ABB RobotStudio station: Apartado4.rspag

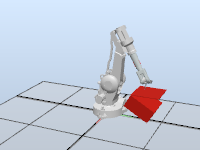
--- station ---
Station Práctica_1_casa (saved by RobotStudio 7.0.8746.631)
Controller IRB_2400_12kg_1.55m
  mechanical unit ROB_1: IRB2400_10_150__02, 6 joints, base frame (0, 0, 0) mm
Layout (positions relative to the parent item):
  - IRB2400_10_150__02 [mechanism, from Robots\IRB2400_10_150_G_02.rslib] at (0, 0, 0) mm; joint values [1.6074, 0.1285, 1.0857, 1.3381, 1.0961, 3.693] (rad or m)
  - Inclinado [part] at (-150, 550, 100) mm, rotated rx 0 ry 30 rz 90 deg
  - Garra_puntero_simple [smart component, from Libraries\Garra_puntero_simple.rslib] at (-97.85, 661.37, 666.74) mm, rotated rx -180 ry 60 rz 0 deg
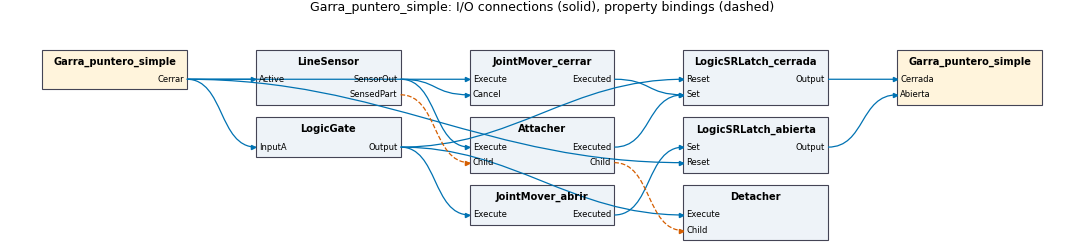
      connections:
        Garra_puntero_simple.Cerrar -> LineSensor.Active
        LineSensor.SensorOut -> Attacher.Execute
        Garra_puntero_simple.Cerrar -> JointMover_cerrar.Execute
        LineSensor.SensorOut -> JointMover_cerrar.Cancel
        Garra_puntero_simple.Cerrar -> LogicGate.InputA
        LogicGate.Output -> Detacher.Execute
        LogicGate.Output -> JointMover_abrir.Execute
        LogicGate.Output -> LogicSRLatch_cerrada.Reset
        LogicSRLatch_cerrada.Output -> Garra_puntero_simple.Cerrada
        JointMover_abrir.Executed -> LogicSRLatch_abierta.Set
        Garra_puntero_simple.Cerrar -> LogicSRLatch_abierta.Reset
        LogicSRLatch_abierta.Output -> Garra_puntero_simple.Abierta
        Attacher.Executed -> LogicSRLatch_cerrada.Set
        JointMover_cerrar.Executed -> LogicSRLatch_cerrada.Set
        LineSensor.SensedPart => Attacher.Child
        Attacher.Child => Detacher.Child
    - LineSensor [smart component, from Components\LineSensor.rslib] at (0, 60, 0) mm
        properties: Start=[0 -0.0595 0.149]; End=[3.45126646034193E-31 -0.0595 0.045]; Radius=0.0001; SensedPart=(none); SensedPoint=[0 0 0]
      - _sensorPart_ [part]
    - Attacher [smart component, from Components\Attacher.rslib]
        properties: Parent=Mecanismo_garra_puntero_simple; Flange=0; Child=(none); Mount=false; Offset=[0 0 0]; Orientation=[0 0 0]
    - Detacher [smart component, from Components\Detacher.rslib]
        properties: Child=Mecanismo_garra_puntero_simple; KeepPosition=true
    - JointMover_cerrar [smart component, from Components\JointMover.rslib]
        properties: Mechanism=Mecanismo_garra_puntero_simple; Relative=false; Duration=0.5; J1=0
    - LogicGate [smart component, from Components\LogicGate.rslib]
        properties: Operator=NOT; Delay=0
    - JointMover_abrir [smart component, from Components\JointMover.rslib]
        properties: Mechanism=Mecanismo_garra_puntero_simple; Relative=false; Duration=0.5; J1=0.06
    - LogicSRLatch_cerrada [smart component, from Components\LogicSRLatch.rslib]
    - LogicSRLatch_abierta [smart component, from Components\LogicSRLatch.rslib]
    - Mecanismo_garra_puntero_simple [mechanism, from Libraries\Garra_puntero_simple.rslib] at (0, 0, 0) mm; joint values [0.06] (rad or m)
Attachment: LineSensor is attached to Mecanismo_garra_puntero_simple / Dedp_1
Attachment: Garra_puntero_simple is attached to IRB2400_10_150__02 / Link6
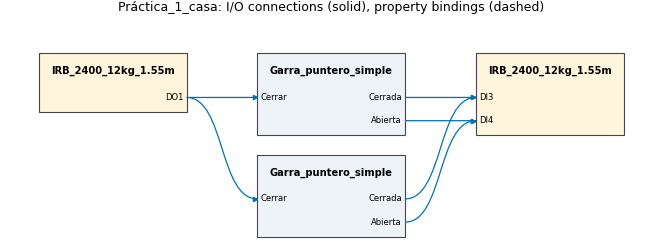
Station logic (signal -> signal, property => property):
  Garra_puntero_simple.Cerrada -> IRB_2400_12kg_1.55m.DI3
  Garra_puntero_simple.Abierta -> IRB_2400_12kg_1.55m.DI4
  IRB_2400_12kg_1.55m.DO1 -> Garra_puntero_simple.Cerrar
  Garra_puntero_simple.Cerrada -> IRB_2400_12kg_1.55m.DI3
  Garra_puntero_simple.Abierta -> IRB_2400_12kg_1.55m.DI4
  IRB_2400_12kg_1.55m.DO1 -> Garra_puntero_simple.Cerrar

--- Backups/IRB_2400_12kg_1.55m/RAPID/TASK1/PROGMOD/Module1.mod ---
MODULE Module1
    PERS tooldata Garra_TCP:=[TRUE,[[0,0,150],[0,1,0,0]],[1,[0,0,10],[1,0,0,0],0,0,0]];
    PERS tooldata Puntero_TCP:=[TRUE,[[150,0,30],[0.707106781,0,-0.707106781,0]],[1,[0,0,10],[1,0,0,0],0,0,0]];
    CONST confdata config_fun:=[0,0,0,0];
    CONST confdata config_fuf:=[0,0,0,1];
    CONST extjoint ejes_externos:=[9E+09,9E+09,9E+09,9E+09,9E+09,9E+09];
    CONST jointtarget casa:=[[0,0,0,0,0,0],ejes_externos];
    CONST num distancia:=150;
    TASK PERS wobjdata plano_trazado:=[FALSE,TRUE,"",[[101.172,952.795,450.836],[2.49104E-07,0,0,1]],[[0,0,0],[1,0,0,0]]];

    VAR intnum emergencia;

    PROC Pinta_cuadrado(robtarget centro, PERS wobjdata objeto_trabajo, PERS tooldata tool)
        VAR robtarget Paprox;
        VAR robtarget P1;
        VAR robtarget P2;
        VAR robtarget P3;
        VAR robtarget P4;

        Paprox:= RelTool (centro, 0, 0, 50);
        MoveJ Paprox, v500, fine, tool\WObj:=objeto_trabajo;

        P1:= RelTool (centro, 50, 50, 0);
        MoveL P1, v500, fine, tool\WObj:=objeto_trabajo;

        P2:= RelTool (centro, 50, -50, 0);
        MoveL P2, v500, fine, tool\WObj:=objeto_trabajo;

        P3:= RelTool (centro, -50, -50, 0);
        MoveL P3, v500, fine, tool\WObj:=objeto_trabajo;

        P4:= RelTool (centro, -50, 50, 0);
        MoveL P4, v500, fine, tool\WObj:=objeto_trabajo;

        !Move to complete square
        MoveL P1, v500, fine, tool\WObj:=objeto_trabajo;

        !Move to approximation position
        MoveL Paprox, v500, fine, tool\WObj:=objeto_trabajo;
    ENDPROC

    PROC Pinta_circunferencia(robtarget centro, PERS wobjdata objeto_trabajo, PERS tooldata tool)
        VAR robtarget Paprox;
        VAR robtarget P1;
        VAR robtarget P2;
        VAR robtarget P3;
        VAR robtarget P4;

        Paprox:= RelTool (centro, 0, 0, 50);
        MoveJ Paprox, v500, fine, tool\WObj:=objeto_trabajo;

        P1:= RelTool (centro, 0, 100*Sqrt(2), 0);
        P2:= RelTool (centro, 100*Sqrt(2), 0, 0);
        P3:= RelTool (centro, 0, -100*Sqrt(2), 0);
        P4:= RelTool (centro, -100*Sqrt(2), 0, 0);

        MoveL P1, v500, fine, tool\WObj:=objeto_trabajo;
        MoveC P2, P3, v500, fine, tool\WObj:=objeto_trabajo;
        MoveC P4, P1, v500, fine, tool\WObj:=objeto_trabajo;

        MoveJ Paprox, v500, fine, tool\WObj:=objeto_trabajo;

	ENDPROC

    PROC cerrar()
        ! Completa el código fuente
    ENDPROC

    PROC abrir()
        ! Completa el código fuente
    ENDPROC


    PROC main()
        VAR robtarget ptest := [[150, 150, 0],[1,0,0,0], config_fun, [0,0,0,0,9E9,9E9] ];
        ptest:= RelTool(ptest, 0, 0, 71\Ry:=30);

        CONNECT emergencia WITH emergency_routine;
        ISignalDI DI3, 1, emergencia;

        MoveAbsJ casa, v1000, fine, Puntero_TCP;
        WHILE DI1=0 DO
            IF DI2=0 THEN
                Pinta_cuadrado ptest, plano_trazado, Puntero_TCP;
            ELSE
                Pinta_circunferencia ptest, plano_trazado, Puntero_TCP;
            ENDIF
        ENDWHILE
        MoveAbsJ casa, v1000, fine, Puntero_TCP;
    ENDPROC

    TRAP emergency_routine
        StopMove \Quick;
        TPWrite "Emergencia, esperando DI3==0";
        WaitDI DI3, 0;
        TPWrite "Reanudando ejecución";
        StartMove;
    ENDTRAP

ENDMODULE

--- Backups/IRB_2400_12kg_1.55m/RAPID/TASK1/SYSMOD/LINKEDM.sys ---
%%%
  VERSION:1
  LANGUAGE:ENGLISH
%%%

MODULE LINKEDM (SYSMODULE)

! FOLLOWER
!     Name of electronically linked follower axis used by operator at teach pendent.
      PERS string l_f_axis_name{5}       :=  ["",  "", "", "", ""];

!     Name of the mechanical unit for follower axis.
      PERS string l_f_mecunt_n{5}  :=  ["", "", "", "", ""];

!     Linked follower axis number in the mechanical unit (first axis in mech. unit is number 1).
      PERS num l_f_axis_no{5}      :=  [0,          0,   0,  0,  0];

! MASTER
!     Name of the mechanical unit for linked master axis.
      PERS string l_m_mecunt_n{5} :=  ["", "", "", "", ""];

!     Linked master axis number in the mechanical unit (first axis in mech. unit is number 1).
!     See axis number table in documentation for different master mechanical units.
      PERS num l_m_axis_no{5}     :=  [0,  0,  0,  0,  0];

! POSITION OFFSET
!     The increase of the allowed offset position between the master and follower
!     positions, used when starting AUTO mode. As soon as the offset is decreased
!     the old configurated parameter is used.
!     Example: 3 => the configurated value of allowed offset is increased 3 times.
      PERS num offset_ratio{5}       :=  [10,  10,   10,  10,  10];

! SPEED RATIO
!     Speed_ratio used in AUTO and JOG modes [ very_slow   slow    normal    fast]
!     Value 1 = max allowed manual speed.
      CONST num speed_ratio {20}      := [0.01, 0.01, 0.01, 0.01, 0.01,
                                          0.05, 0.05, 0.05, 0.05, 0.05,
                                          0.20, 0.20, 0.20, 0.20, 0.20,
                                          1.00, 1.00, 1.00, 1.00, 1.00];

! STEP SIZE
!     Displacement position used in JOG mode for each activation of positive or
!     negative movement.                  [very_short    short   normal   long]
!     Unit degees or meter.
      CONST num displacement {20}     := [0.001, 0.001, 0.001, 0.001, 0.001,
                                          0.005, 0.005, 0.005, 0.005, 0.005,
                                          0.020, 0.020, 0.020, 0.020, 0.020,
                                          0.100, 0.100, 0.100, 0.100, 0.100];


!-------------------------------------------------------------
 PROC Linked_m ()
      Linked_m_exe ;
 ENDPROC
ENDMODULE

--- Backups/IRB_2400_12kg_1.55m/SYSPAR/EIO.cfg ---
EIO:CFG_1.0:6:1::
#
EIO_SIGNAL:

      -Name "DI1" -SignalType "DI"

      -Name "DI2" -SignalType "DI"

      -Name "DO1" -SignalType "DO"

      -Name "DO2" -SignalType "DO"

      -Name "DI3" -SignalType "DI"

      -Name "DI4" -SignalType "DI"

      -Name "DI5" -SignalType "DI"

      -Name "DO3" -SignalType "DO"

      -Name "DO4" -SignalType "DO"

      -Name "DO5" -SignalType "DO"
